{attribute 'strict'}
TYPE E_CognexCameraPutTimeoutStatus :
(
	WAITING_FOR_STATUS_CODE										:= 2,	
	THE_COMMAND_WAS_EXECUTED_SUCCESSFULLY						:= 1,
	UNRECOGNIZED_COMMAND 										:= 0,
	THE_INPUT_IS_INVALID_OR_HAS_EXCEEDED_15_BYTES_IN_LENGTH		:= -1,
	USER_DOES_NOT_HAVE_FULL_ACCESS	 							:= -6
);
END_TYPE

(* stored: Version 1.1.0.1, ProductVersion 3.1.4024.9
   DUT E_CognexCameraPutTimeoutStatus: Id {3da835d3-9c7a-406f-a7d2-461d23f775c5} *)
